{attribute addProperty BoxType "EK1960-0000-0019"}
{attribute addProperty Id "OutputsOutputs_B00B49A922428"}
{attribute addProperty CRC "986779022"}
{attribute addProperty SizeInBites "224"}
{attribute addProperty SizeInBytes "28"}
TYPE Module_2_FSOUT_3AD10D8E :
STRUCT
	{attribute addProperty Name "Outputs"}
	Outputs  : Outputs_B00B49A9;
END_STRUCT
END_TYPE

(* stored: Version 1.2.0.0, ProductVersion 3.1.4024.9
   DUT Module_2_FSOUT_3AD10D8E: Id {539eacec-9af9-49e0-b5d6-7f1404dc23f8} *)
